TYPE ST_Syntax_PointerRef :
    STRUCT
        pData : POINTER TO INT;
        rItem : REFERENCE TO INT;
    END_STRUCT
END_TYPE

(* stored: Version 1.1.0.1, ProductVersion 3.1.4024.16
   DUT ST_Syntax_PointerRef: Id {8801a84f-2908-4435-9139-4ab69390263b} *)
